Staubli VAL3: OnF1.pgx

program OnF1()
  local bool l_bRes
  local string l_sYesNo[2]
begin
  //单一路径转化
  //
  //检查文件是否已经存在
  call chkIsFileExsit(sItem,sOutputFolder,l_bRes)
  //存在，询问
  if l_bRes
    l_sYesNo[0]="是"
    l_sYesNo[1]="否"
    call user:yes_no("文件已存在，是否覆盖?",l_sYesNo,l_bRes)
    bUserRefresh=true
    if !l_bRes
      return
    else
      $delete(sOutputFolder+sItem)
    endIf
  endIf
  //

  //转换文件
  call OnePathConvert(sFolder,sItem,sOutputFolder,l_bRes)
  if l_bRes
    popUpMsg("转换完成")
  else
    popUpMsg("文件转换失败!")
  endIf
end
